// TIA Portal project "Schrittkette_0" (V20)

(* hardware
DEVICE "S7-1500/ET200MP-Station_1"  S7-1500 station
   slot 0: "Profilschiene_0"  Rack  6ES7 590-1***0-0AA0
   slot 1: "PLC_1"  CPU 1513-1 PN  6ES7 513-1AM03-0AB0  V4.0
      slot 3: "CPU-Display_1"  6ES7591-1AA00-0AA0
      slot 32768: "PROFINET-Schnittstelle_1"  X1
         slot 32769: "Port_1"  X1 P1
         slot 32770: "Port_2"  X1 P2
      slot 34817: "Virtual CP interface port_1"  Virtual CP interface port  Virtual CP interface port FW V4.0
   slot 2: "DI 16x24VDC BA_1"  DI 16x24VDC BA  6ES7 521-1BH10-0AA0  V1.1
   slot 3: "DQ 16x24VDC/0.5A ST_1"  DQ 16x24VDC/0.5A ST  6ES7 522-1BH00-0AB0  V2.0
   slot 4: "AI 8xU/I/R/RTD BA_2"  AI 8xU/I/R/RTD BA  6ES7 531-7QF00-0AB0  V1.0
   slot 5: "AQ 8xU/I HS_2"  AQ 8xU/I HS  6ES7 532-5HF00-0AB0  V2.2
*)

// ===== PLC "PLC_1"  CPU 1513-1 PN =====

VAR_GLOBAL   // PLC tag table "Eingaenge"
   "S1" AT %I0.0 : Bool;   // Start Taster
   "S2" AT %I0.1 : Bool;   // Stop Taster
   "S3" AT %I0.2 : Bool;   // Reset
   "2B1" AT %I0.3 : Bool;   // Sensor Produkt an Stanze
   "3B1" AT %I0.4 : Bool;   // Sensor Produkt am Pusher
   "1B1" AT %I0.5 : Bool;   // Sensor Einlauf (Start)
   "2B2" AT %I0.6 : Bool;   // Stanze unten
   "3B2" AT %I0.7 : Bool;   // Pusher hinten
   "3B3" AT %I1.0 : Bool;   // Pusher vorne
END_VAR

VAR_GLOBAL   // PLC tag table "Ausgaenge"
   "M1" AT %Q0.0 : Bool;   // Motor Förderer
   "M2" AT %Q0.1 : Bool;   // Stanze
   "M3" AT %Q0.2 : Bool;   // Pusher
   "H1" AT %Q0.3 : Bool;   // Leuchte Anlage Ein
   "H2" AT %Q0.4 : Bool;   // Leuchte Anlage Aus
   "H3" AT %Q0.5 : Bool;   // Meldeleuchte gelb
END_VAR

DATA_BLOCK "Anlagedaten"   // DB1
{ S7_Optimized_Access := 'TRUE' }
VERSION : 0.1
   VAR
      Anlage : Struct
         Start : Bool;
         Stopp : Bool;
         Reset : Bool;
         Aktiv : Bool;
      END_STRUCT;
      Betriebsdaten : Struct
         Schritt_aktiv : Bool;
         Schritt : Array[1..10] of Bool;
         Sensoren : Struct
            Einlauf : Bool;
            Produkt_bei_Stanze : Bool;
            Stanze_unten : Bool;
            Produkt_bei_Pusher : Bool;
            Pusher_hinten : Bool;
            Pusher_vorne : Bool;
         END_STRUCT;
         Aktoren : Struct
            Foerderer : Bool;
            Stanze : Bool;
            Pusher : Bool;
            Leuchten : Struct
               Gruen : Bool;
               Rot : Bool;
               Gelb : Bool;
            END_STRUCT;
         END_STRUCT;
         Stanze_Daten : IEC_TIMER;
      END_STRUCT;
   END_VAR
BEGIN
END_DATA_BLOCK

FUNCTION "Anlagensteuerung" : Void   // FC1, FBD
{ S7_Optimized_Access := 'TRUE' }
VERSION : 0.1
BEGIN

REGION Network 1
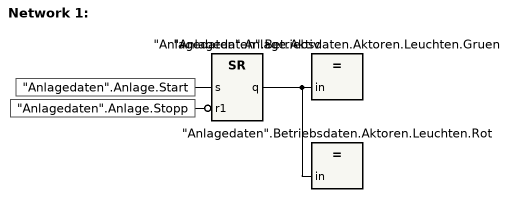
   IF "Anlagedaten".Anlage.Start THEN
       "Anlagedaten".Anlage.Aktiv := TRUE;   // SR flip-flop
   END_IF;
   IF NOT "Anlagedaten".Anlage.Stopp THEN "Anlagedaten".Anlage.Aktiv := FALSE; END_IF;
   "Anlagedaten".Betriebsdaten.Aktoren.Leuchten.Gruen := "Anlagedaten".Anlage.Aktiv;
   "Anlagedaten".Betriebsdaten.Aktoren.Leuchten.Rot := "Anlagedaten".Anlage.Aktiv;
END_REGION
END_FUNCTION

FUNCTION "Schrittkette" : Void   // FC2, FBD
{ S7_Optimized_Access := 'TRUE' }
VERSION : 0.1
   VAR_IN_OUT
      Stanze_Verzoegerung : TON_TIME;
   END_VAR
BEGIN

REGION Network 1
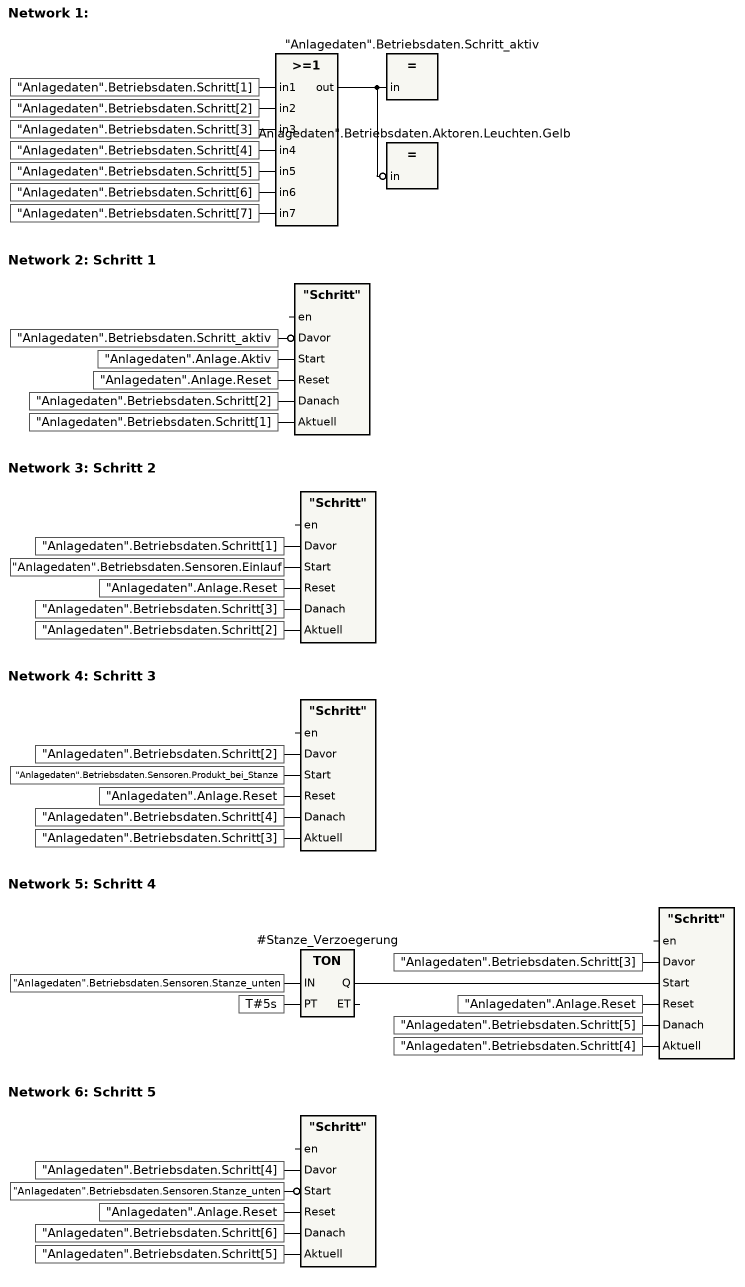
   "Anlagedaten".Betriebsdaten.Schritt_aktiv := "Anlagedaten".Betriebsdaten.Schritt[1] OR "Anlagedaten".Betriebsdaten.Schritt[2] OR "Anlagedaten".Betriebsdaten.Schritt[3] OR "Anlagedaten".Betriebsdaten.Schritt[4] OR "Anlagedaten".Betriebsdaten.Schritt[5] OR "Anlagedaten".Betriebsdaten.Schritt[6] OR "Anlagedaten".Betriebsdaten.Schritt[7];
   "Anlagedaten".Betriebsdaten.Aktoren.Leuchten.Gelb := NOT "Anlagedaten".Betriebsdaten.Schritt_aktiv;
END_REGION

REGION Network 2: Schritt 1
   "Schritt"(Davor := NOT "Anlagedaten".Betriebsdaten.Schritt_aktiv,
             Start := "Anlagedaten".Anlage.Aktiv,
             Reset := "Anlagedaten".Anlage.Reset,
             Danach := "Anlagedaten".Betriebsdaten.Schritt[2],
             Aktuell := "Anlagedaten".Betriebsdaten.Schritt[1]);
END_REGION

REGION Network 3: Schritt 2
   "Schritt"(Davor := "Anlagedaten".Betriebsdaten.Schritt[1],
             Start := "Anlagedaten".Betriebsdaten.Sensoren.Einlauf,
             Reset := "Anlagedaten".Anlage.Reset,
             Danach := "Anlagedaten".Betriebsdaten.Schritt[3],
             Aktuell := "Anlagedaten".Betriebsdaten.Schritt[2]);
END_REGION

REGION Network 4: Schritt 3
   "Schritt"(Davor := "Anlagedaten".Betriebsdaten.Schritt[2],
             Start := "Anlagedaten".Betriebsdaten.Sensoren.Produkt_bei_Stanze,
             Reset := "Anlagedaten".Anlage.Reset,
             Danach := "Anlagedaten".Betriebsdaten.Schritt[4],
             Aktuell := "Anlagedaten".Betriebsdaten.Schritt[3]);
END_REGION

REGION Network 5: Schritt 4
   #Stanze_Verzoegerung(IN := "Anlagedaten".Betriebsdaten.Sensoren.Stanze_unten, PT := T#5s);   // TON
   "Schritt"(Davor := "Anlagedaten".Betriebsdaten.Schritt[3],
             Start := #Stanze_Verzoegerung.Q,
             Reset := "Anlagedaten".Anlage.Reset,
             Danach := "Anlagedaten".Betriebsdaten.Schritt[5],
             Aktuell := "Anlagedaten".Betriebsdaten.Schritt[4]);
END_REGION

REGION Network 6: Schritt 5
   "Schritt"(Davor := "Anlagedaten".Betriebsdaten.Schritt[4],
             Start := NOT "Anlagedaten".Betriebsdaten.Sensoren.Stanze_unten,
             Reset := "Anlagedaten".Anlage.Reset,
             Danach := "Anlagedaten".Betriebsdaten.Schritt[6],
             Aktuell := "Anlagedaten".Betriebsdaten.Schritt[5]);
END_REGION

REGION Network 7: Schritt 6
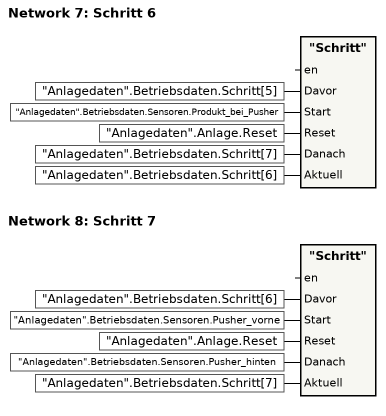
   "Schritt"(Davor := "Anlagedaten".Betriebsdaten.Schritt[5],
             Start := "Anlagedaten".Betriebsdaten.Sensoren.Produkt_bei_Pusher,
             Reset := "Anlagedaten".Anlage.Reset,
             Danach := "Anlagedaten".Betriebsdaten.Schritt[7],
             Aktuell := "Anlagedaten".Betriebsdaten.Schritt[6]);
END_REGION

REGION Network 8: Schritt 7
   "Schritt"(Davor := "Anlagedaten".Betriebsdaten.Schritt[6],
             Start := "Anlagedaten".Betriebsdaten.Sensoren.Pusher_vorne,
             Reset := "Anlagedaten".Anlage.Reset,
             Danach := "Anlagedaten".Betriebsdaten.Sensoren.Pusher_hinten,
             Aktuell := "Anlagedaten".Betriebsdaten.Schritt[7]);
END_REGION
END_FUNCTION

FUNCTION "Schritt" : Void   // FC3, FBD
{ S7_Optimized_Access := 'TRUE' }
VERSION : 0.1
   VAR_INPUT
      Davor : Bool;
      Start : Bool;
      Reset : Bool;
      Danach : Bool;
   END_VAR
   VAR_IN_OUT
      Aktuell : Bool;
   END_VAR
BEGIN

REGION Network 1
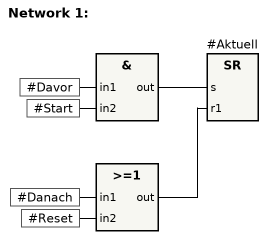
   IF #Davor AND #Start THEN
       #Aktuell := TRUE;   // SR flip-flop
   END_IF;
   IF #Danach OR #Reset THEN #Aktuell := FALSE; END_IF;
END_REGION
END_FUNCTION

FUNCTION "Ansteuerung_Maschinen" : Void   // FC4, FBD
{ S7_Optimized_Access := 'TRUE' }
VERSION : 0.1
BEGIN

REGION Network 1
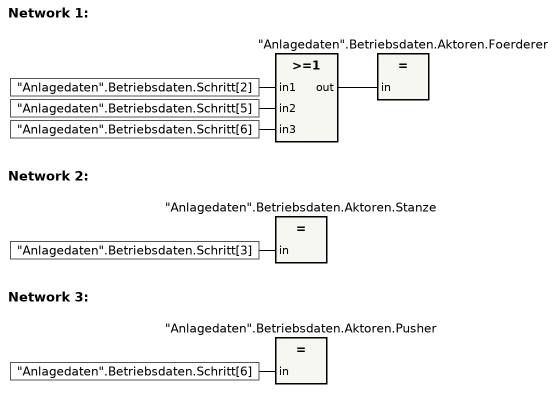
   "Anlagedaten".Betriebsdaten.Aktoren.Foerderer := "Anlagedaten".Betriebsdaten.Schritt[2] OR "Anlagedaten".Betriebsdaten.Schritt[5] OR "Anlagedaten".Betriebsdaten.Schritt[6];
END_REGION

REGION Network 2
   "Anlagedaten".Betriebsdaten.Aktoren.Stanze := "Anlagedaten".Betriebsdaten.Schritt[3];
END_REGION

REGION Network 3
   "Anlagedaten".Betriebsdaten.Aktoren.Pusher := "Anlagedaten".Betriebsdaten.Schritt[6];
END_REGION
END_FUNCTION

FUNCTION "EA" : Void   // FC100, FBD
{ S7_Optimized_Access := 'TRUE' }
VERSION : 0.1
BEGIN

REGION Network 1
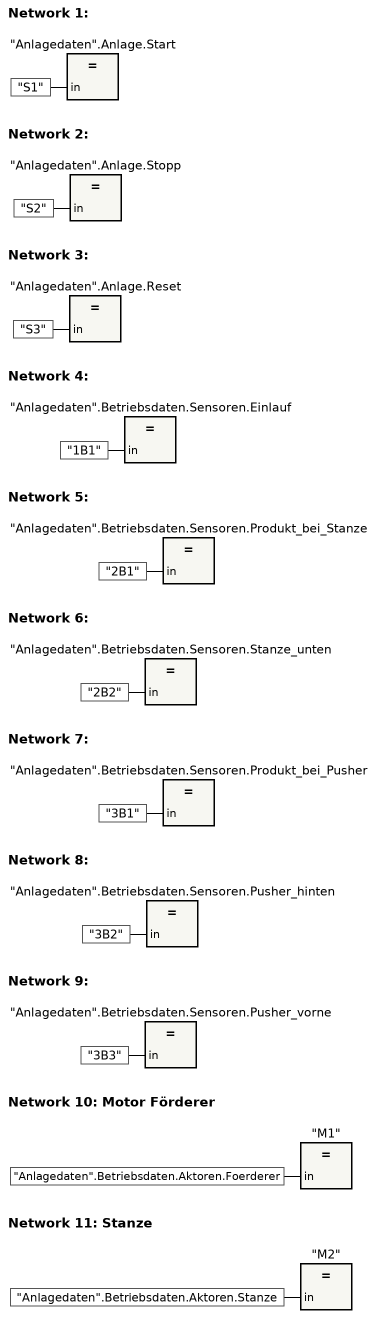
   "Anlagedaten".Anlage.Start := "S1";
END_REGION

REGION Network 2
   "Anlagedaten".Anlage.Stopp := "S2";
END_REGION

REGION Network 3
   "Anlagedaten".Anlage.Reset := "S3";
END_REGION

REGION Network 4
   "Anlagedaten".Betriebsdaten.Sensoren.Einlauf := "1B1";
END_REGION

REGION Network 5
   "Anlagedaten".Betriebsdaten.Sensoren.Produkt_bei_Stanze := "2B1";
END_REGION

REGION Network 6
   "Anlagedaten".Betriebsdaten.Sensoren.Stanze_unten := "2B2";
END_REGION

REGION Network 7
   "Anlagedaten".Betriebsdaten.Sensoren.Produkt_bei_Pusher := "3B1";
END_REGION

REGION Network 8
   "Anlagedaten".Betriebsdaten.Sensoren.Pusher_hinten := "3B2";
END_REGION

REGION Network 9
   "Anlagedaten".Betriebsdaten.Sensoren.Pusher_vorne := "3B3";
END_REGION

REGION Network 10: Motor Förderer
   "M1" := "Anlagedaten".Betriebsdaten.Aktoren.Foerderer;
END_REGION

REGION Network 11: Stanze
   "M2" := "Anlagedaten".Betriebsdaten.Aktoren.Stanze;
END_REGION

REGION Network 12: Pusher
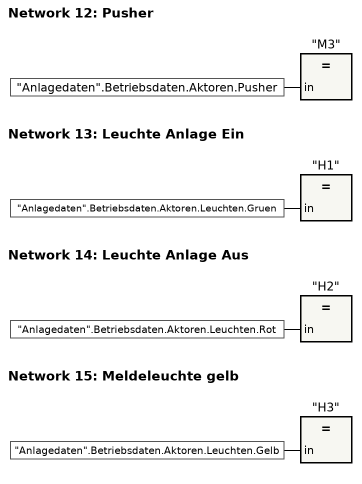
   "M3" := "Anlagedaten".Betriebsdaten.Aktoren.Pusher;
END_REGION

REGION Network 13: Leuchte Anlage Ein
   "H1" := "Anlagedaten".Betriebsdaten.Aktoren.Leuchten.Gruen;
END_REGION

REGION Network 14: Leuchte Anlage Aus
   "H2" := "Anlagedaten".Betriebsdaten.Aktoren.Leuchten.Rot;
END_REGION

REGION Network 15: Meldeleuchte gelb
   "H3" := "Anlagedaten".Betriebsdaten.Aktoren.Leuchten.Gelb;
END_REGION
END_FUNCTION

ORGANIZATION_BLOCK "Main"   // OB1, FBD, ProgramCycle
TITLE = "Main Program Sweep (Cycle)"
{ S7_Optimized_Access := 'TRUE' }
VERSION : 0.1
   VAR_INPUT
      Initial_Call : Bool;   // Initial call of this OB
      Remanence : Bool;   // =True, if remanent data are available
   END_VAR
BEGIN

REGION Network 1
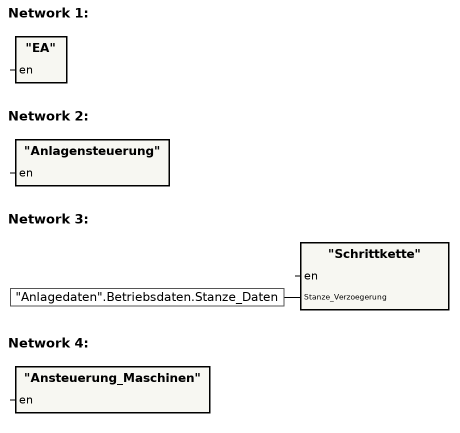
   "EA"();
END_REGION

REGION Network 2
   "Anlagensteuerung"();
END_REGION

REGION Network 3
   "Schrittkette"(Stanze_Verzoegerung := "Anlagedaten".Betriebsdaten.Stanze_Daten);
END_REGION

REGION Network 4
   "Ansteuerung_Maschinen"();
END_REGION
END_ORGANIZATION_BLOCK